// TIA Portal V16 export
// export: Created 2022-07-21T09:35:15.9930239Z, ExportSetting WithDefaults, DisplayName Totally Integrated Automation Portal, DisplayVersion V16 Update 4, DisplayName TIA Portal Version Control Interface, DisplayVersion V16 Update 2, DisplayName TIA Portal Openness, DisplayVersion V16 Update 4, DisplayName SINAMICS Startdrive Advanced, DisplayVersion V16 Update 5, DisplayName SINAMICS Startdrive G130, G150, S120, S150, SINAMICS MV, S210, DisplayVersion V16 Update 5, DisplayName SINAMICS Startdrive G110M, G120, G120C, G120D, G120P, G115D, DisplayVersion V16 Update 5, DisplayName STEP 7 Professional, DisplayVersion V16 Update 4, DisplayName STEP 7 Safety, DisplayVersion V16, DisplayName WinCC Advanced, DisplayVersion V16 Update 4
FUNCTION_BLOCK "fbMessageWarning"   // FB52, LAD
TITLE = Warning handling / Obsługa ostrzeżeń
{ S7_Optimized_Access := 'TRUE' }
VERSION : 0.1
// stored: AutoNumber true, IsIECCheckEnabled true, IsRetainMemResEnabled false, MemoryReserve 100, SetENOAutomatically false, UDAEnableTagReadback false
   VAR_INPUT
      inEnable { ExternalAccessible := 'False'; ExternalVisible := 'False'; ExternalWritable := 'False'} : Bool;   // Zezwolenie / Permission
      inFbSignalOk { ExternalAccessible := 'False'; ExternalVisible := 'False'; ExternalWritable := 'False'} : Bool;   // Sygnał ok / Signal OK
      inDelaySignalOn { ExternalAccessible := 'False'; ExternalVisible := 'False'; ExternalWritable := 'False'} : Time;   // Opóźnienie ustawienia sygnału wejściowego / delay input signal set
      inDelaySignalOff { ExternalAccessible := 'False'; ExternalVisible := 'False'; ExternalWritable := 'False'} : Time;   // Opóźnienie wyłączenia sygnału wejsciowego / delay input signal reset
   END_VAR
   VAR_OUTPUT
      ouMessage { ExternalAccessible := 'False'; ExternalVisible := 'False'; ExternalWritable := 'False'} : Bool;   // Wygenerowany błąd / Generated error
   END_VAR
   VAR
      sMessage { ExternalAccessible := 'False'; ExternalVisible := 'False'; ExternalWritable := 'False'; S7_SetPoint := 'True'} : "fbMessageHandlingDelayed";
   END_VAR
BEGIN

REGION Network 1: Error handling / Obsługa błędów
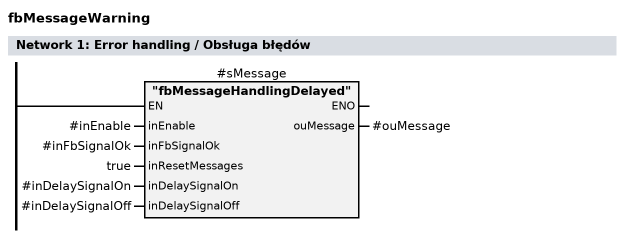
   RUNG wire#powerrail
      #sMessage(inEnable := #inEnable, inFbSignalOk := #inFbSignalOk, inResetMessages := true, inDelaySignalOn := #inDelaySignalOn, inDelaySignalOff := #inDelaySignalOff, ouMessage => #ouMessage)
   END_RUNG
   // the same network as SCL:
   #sMessage(inEnable := #inEnable,   // "fbMessageHandlingDelayed"
             inFbSignalOk := #inFbSignalOk,
             inResetMessages := true,
             inDelaySignalOn := #inDelaySignalOn,
             inDelaySignalOff := #inDelaySignalOff,
             ouMessage => #ouMessage);
END_REGION
END_FUNCTION_BLOCK
